{attribute 'linkalways'} 
{attribute 'no_explicit_call' := 'This FB is a CLASS and must be accessed using methods or properties'}
{attribute 'enable_dynamic_creation'}
FUNCTION_BLOCK FINAL GE_ULINT EXTENDS Node
VAR
	in1 : _ULINT(0);
	in2 : _ULINT(0);
	out : _BOOL(FALSE);
END_VAR

METHOD PUBLIC Clone : I_Node
VAR
	pNode : POINTER TO GE_ULINT;
END_VAR
pNode := __NEW(GE_ULINT);
Clone := pNode^;
END_METHOD

METHOD FB_init : BOOL
VAR_INPUT
	bInitRetains : BOOL; // if TRUE, the retain variables are initialized (warm start / cold start)
	bInCopyCode : BOOL;  // if TRUE, the instance afterwards gets moved into the copy code (online change)
END_VAR
AddInput('in1',THIS^.in1);
AddInput('in2',THIS^.in2);
AddOutput('out', THIS^.out);
END_METHOD

METHOD PROTECTED OnExecute
VAR
END_VAR
out.Value := in1.Value >= in2.Value;
END_METHOD

END_FUNCTION_BLOCK

(* stored: Version 1.1.0.1, ProductVersion 3.1.4024.15
   POU GE_ULINT: Id {01a3c80b-80f7-4d7b-a48b-f7619fd75bdd}, SpecialFunc None
   Folder Constructor: Id {bc7c9146-9180-4809-b09a-762097b22dfb}
   Method Clone: Id {73a1ed1c-4e19-49a6-b2dc-d5902f5c3515}
   Method FB_init: Id {bf4e3f6f-6a22-4c1c-ae7b-c6c254f95b9f}
   Method OnExecute: Id {20e31b80-887a-4d7a-af16-c17d7fa521b4} *)
